(* IEC 61131-3 sources: repolevel_ST_code_completion/real_groud_truth最新/repoeval_core/readful_result, 2 files *)

(* ---- CommandExecutor.st ---- *)
VAR
	direct		:TargetDirect;	//方向
END_VAR

CASE direct OF
	TargetDirect.extend:
		CASE level OF
			1:
				gController.grd[idx].extendPercent := REAL_TO_WORD(percent * 65535 / 100);
				gController.grd[idx].retractPercent := 0;
			2:
				gController.sky[idx].extendPercent := REAL_TO_WORD(percent * 65535 / 100);
				gController.sky[idx].retractPercent := 0;
		END_CASE
	TargetDirect.retract:
		CASE level OF
			1:
				gController.grd[idx].extendPercent := 0;
				gController.grd[idx].retractPercent := REAL_TO_WORD(ABS(percent) * 65535 / 100);
			2:
				gController.sky[idx].extendPercent := 0;
				gController.sky[idx].retractPercent := REAL_TO_WORD(ABS(percent) * 65535 / 100);
		END_CASE
	TargetDirect.stop:
		CASE level OF
			1:
				gController.grd[idx].extendPercent := 0;
				gController.grd[idx].retractPercent := 0;
			2:
				gController.sky[idx].extendPercent := 0;
				gController.sky[idx].retractPercent := 0;
		END_CASE
END_CASE

(* ---- CommandExecutor0.st ---- *)
VAR
END_VAR

CASE direct OF
	TargetDirect.Extend:
		CASE level OF
			1:
				gController.grd[idx].extendPercent := REAL_TO_WORD(percent * 65535 / 100);
				gController.grd[idx].retractPercent := 0;
			2:
				gController.sky[idx].extendPercent := REAL_TO_WORD(percent * 65535 / 100);
				gController.sky[idx].retractPercent := 0;
		END_CASE;
	TargetDirect.Retract:
		CASE level OF
			1:
				gController.grd[idx].extendPercent := 0;
				gController.grd[idx].retractPercent := REAL_TO_WORD(percent * 65535 / 100);
			2:
				gController.sky[idx].extendPercent := 0;
				gController.sky[idx].retractPercent := REAL_TO_WORD(percent * 65535 / 100);
		END_CASE;
END_CASE;
